// TIA Portal project "TEST_Project" (V16)

(* hardware
DEVICE "S7-1200 station_1"  S7-1200 Station
   slot 0: "Rack_0"  S7-1200 Rack  Rack  V1.0
   slot 1: "PLC_1"  CPU 1212C AC/DC/Rly  6ES7 212-1BE40-0XB0  V4.2
   slot 2: "AI 4x13BIT/AQ 2x14BIT_1"  6ES7 234-4HE32-0XB0  V2.1
*)

// ===== PLC "PLC_1"  CPU 1212C AC/DC/Rly =====

VAR_GLOBAL   // PLC tag table "Default tag table"
   "Level Tank 1" AT %IW96 : Int;
   "Level Tank 2" AT %IW66 : Int;
   "StartPump1" AT %I0.0 : Bool;
   "Stop1" AT %I0.1 : Bool;
   "StartPump2" AT %I0.2 : Bool;
   "Stop2" AT %I0.3 : Bool;
   "Level Tank 3" AT %IW96 : Int;
   "Level Tank 4" AT %IW98 : Int;
   "Pump1" AT %Q0.0 : Bool;
   "Pump2" AT %Q0.1 : Bool;
   "Tag_45" AT %QW96 : Int;
   "FV2 Write" AT %QW98 : Int;
   "Level Tank 1 Memory" AT %MD50 : Real;
   "Level Tank 2 Memory" AT %MD58 : Real;
   "FV1 Wirite" AT %MD20 : Real;
   "FV1 Real" AT %MD24 : Real;
   "FV2 Memory" AT %MD28 : Real;
   "FV2 Real" AT %MD32 : Real;
   "Clock_Byte" AT %MB0 : Byte;
   "Clock_10Hz" AT %M0.0 : Bool;
   "Clock_5Hz" AT %M0.1 : Bool;
   "Clock_2.5Hz" AT %M0.2 : Bool;
   "Clock_2Hz" AT %M0.3 : Bool;
   "Clock_1.25Hz" AT %M0.4 : Bool;
   "Clock_1Hz" AT %M0.5 : Bool;
   "Clock_0.625Hz" AT %M0.6 : Bool;
   "Clock_0.5Hz" AT %M0.7 : Bool;
   "Level Tank 3 Memory" AT %MD66 : Real;
   "Level Tank 4 Memory" AT %MD74 : Real;
   "Tag_2" AT %MD22 : Real;
   "Tag_3" AT %IW64 : Int;
   "Tag_4" AT %IW68 : Int;
   "Tag_5" AT %MD110 : DWord;
   "Tag_6" AT %MD4 : DWord;
   "Tag_7" AT %QW80 : Word;
   "Tag_1" AT %MW10 : Int;
   "Tag_8" AT %MD36 : Real;
   "Tag_9" AT %MD14 : Real;
   "Tag_10" AT %MD18 : DWord;
   "Tag_11" AT %MD10 : DWord;
END_VAR

ORGANIZATION_BLOCK "Main"   // OB1, LAD, ProgramCycle
TITLE = "Main Program Sweep (Cycle)"
{ S7_Optimized_Access := 'TRUE' }
VERSION : 0.1
   VAR_INPUT
      Initial_Call : Bool;   // Initial call of this OB
      Remanence : Bool;   // =True, if remanent data are available
   END_VAR
BEGIN

REGION Network 1
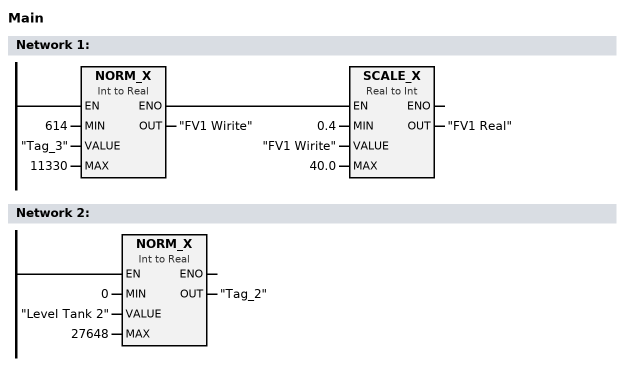
   RUNG wire#powerrail
      { S7_Templates := "[SrcType := Int, DestType := Real]" } Normalize(min := 614, value := "Tag_3", max := 11330, out => "FV1 Wirite")
      { S7_Templates := "[SrcType := Real, DestType := Int]" } Scale(min := 0.4, value := "FV1 Wirite", max := 40.0, out => "FV1 Real")
   END_RUNG
   // the same network as SCL:
   "FV1 Wirite" := NORM_X(MIN := 614, VALUE := "Tag_3", MAX := 11330);
   "FV1 Real" := SCALE_X(MIN := 0.4, VALUE := "FV1 Wirite", MAX := 40.0);
END_REGION

REGION Network 2
   RUNG wire#powerrail
      { S7_Templates := "[SrcType := Int, DestType := Real]" } Normalize(min := 0, value := "Level Tank 2", max := 27648, out => "Tag_2")
   END_RUNG
   // the same network as SCL:
   "Tag_2" := NORM_X(MIN := 0, VALUE := "Level Tank 2", MAX := 27648);
END_REGION
END_ORGANIZATION_BLOCK